// TIA Portal project "OEE_REAL_TIME" (V19)

(* hardware
DEVICE "S7-1200 station_1"  S7-1200 Station
   slot 0: "Rack_0"  Rack  V1.0
   slot 1: "OEE_REAL_TIME"  CPU 1214C DC/DC/DC  6ES7 214-1AG40-0XB0  V4.1
*)

// ===== PLC "OEE_REAL_TIME"  CPU 1214C DC/DC/DC =====
// protected blocks, not shown: "FB_OEE_Calculator"

VAR_GLOBAL   // PLC tag table "Default tag table"
   "Tag_1" AT %M0.0 : Bool;
   "Tag_2" AT %M0.1 : Bool;
   "Tag_3" AT %M0.2 : Bool;
   "Tag_4" AT %M0.3 : Bool;
   "Tag_5" AT %M0.4 : Bool;
END_VAR

DATA_BLOCK "FB_OEE_Calculator_DB"   // DB6
{ S7_Optimized_Access := 'TRUE' }
VERSION : 0.1
// stored: InstanceOfName FB_OEE_Calculator
"FB_OEE_Calculator"
BEGIN
END_DATA_BLOCK

ORGANIZATION_BLOCK "Main"   // OB1, LAD, ProgramCycle
TITLE = "Main Program Sweep (Cycle)"
{ S7_Optimized_Access := 'TRUE' }
VERSION : 0.1
   VAR_INPUT
      Initial_Call : Bool;   // Initial call of this OB
      Remanence : Bool;   // =True, if remanent data are available
   END_VAR
   VAR_TEMP
      "CYCLE TIME" : Real;
      PERFORMANCE : Real;
      QUALIDADE : Real;
      DISPONIBILIDADE : Real;
      OEE : Real;
   END_VAR
BEGIN

REGION Network 1
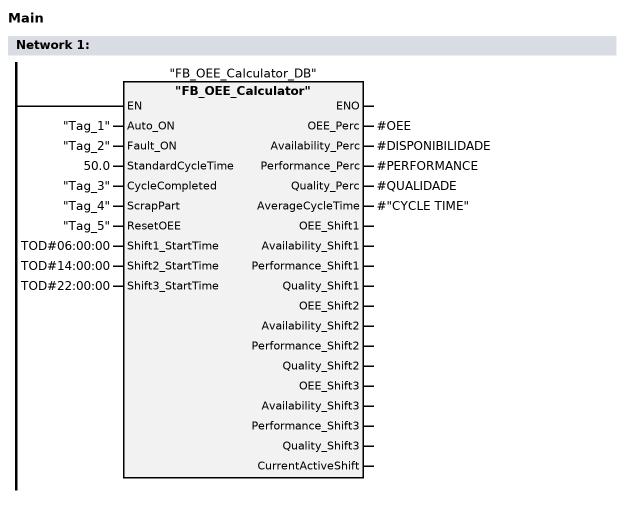
   RUNG wire#powerrail
      "FB_OEE_Calculator_DB"(Auto_ON := "Tag_1", Fault_ON := "Tag_2", StandardCycleTime := 50.0, CycleCompleted := "Tag_3", ScrapPart := "Tag_4", ResetOEE := "Tag_5", Shift1_StartTime := TOD#06:00:00, Shift2_StartTime := TOD#14:00:00, Shift3_StartTime := TOD#22:00:00, OEE_Perc => #OEE, Availability_Perc => #DISPONIBILIDADE, Performance_Perc => #PERFORMANCE, Quality_Perc => #QUALIDADE, AverageCycleTime => #"CYCLE TIME", OEE_Shift1 =>, Availability_Shift1 =>, Performance_Shift1 =>, Quality_Shift1 =>, OEE_Shift2 =>, Availability_Shift2 =>, Performance_Shift2 =>, Quality_Shift2 =>, OEE_Shift3 =>, Availability_Shift3 =>, Performance_Shift3 =>, Quality_Shift3 =>, CurrentActiveShift =>)
   END_RUNG
   // the same network as SCL:
   "FB_OEE_Calculator_DB"(Auto_ON := "Tag_1",   // "FB_OEE_Calculator"
                          Fault_ON := "Tag_2",
                          StandardCycleTime := 50.0,
                          CycleCompleted := "Tag_3",
                          ScrapPart := "Tag_4",
                          ResetOEE := "Tag_5",
                          Shift1_StartTime := TOD#06:00:00,
                          Shift2_StartTime := TOD#14:00:00,
                          Shift3_StartTime := TOD#22:00:00,
                          OEE_Perc => #OEE,
                          Availability_Perc => #DISPONIBILIDADE,
                          Performance_Perc => #PERFORMANCE,
                          Quality_Perc => #QUALIDADE,
                          AverageCycleTime => #"CYCLE TIME");
END_REGION
END_ORGANIZATION_BLOCK